FUNCTION FC_GetLocalDateAndTimeString : T_SHORT_STR		// Returns the local date and time as string,  eg. '27:05:2019 15:58:40:302'. Use E_REGIO_SELECTION at FB_CycleStart for a different format.

FC_GetLocalDateAndTimeString := IING.localDateAndTimeString;

END_FUNCTION

(* stored: Version 1.1.0.1, ProductVersion 3.1.4026.18
   POU FC_GetLocalDateAndTimeString: Id {cbe7610b-d777-46a7-a715-09a2a480dd71}, SpecialFunc None *)
